Fanuc KAREL source: kt00036.KL

PROGRAM KT00036
%NOLOCKGROUP
VAR
I1:INTEGER;R2:REAL;OUT:REAL
BEGIN
--
--
I1=2
R2=3.0
OUT=(I1-R2)
END KT00036
